(* IEC 61131-3 sources: CodesysTest/alpha/export/FBs/Components/MonostableMultivibratorFB.pou, 1 file *)

(* ---- ManualOff.m.st ---- *)
(*#-#-#-#-#-#-#-#-#-#---Declaration---#-#-#-#-#-#-#-#-#-#-#-#-#*)

METHOD ManualOff : BOOL
VAR_INPUT
END_VAR
(*#-#-#-#-#-#-#-#-#-#---Implementation---#-#-#-#-#-#-#-#-#-#-#-#-#*)

_manualOn := FALSE;
_manualOff := TRUE;
